// Mitsubishi GX Works2 project: msp_1   PLC: Q03UDV

PROGRAM MAIN
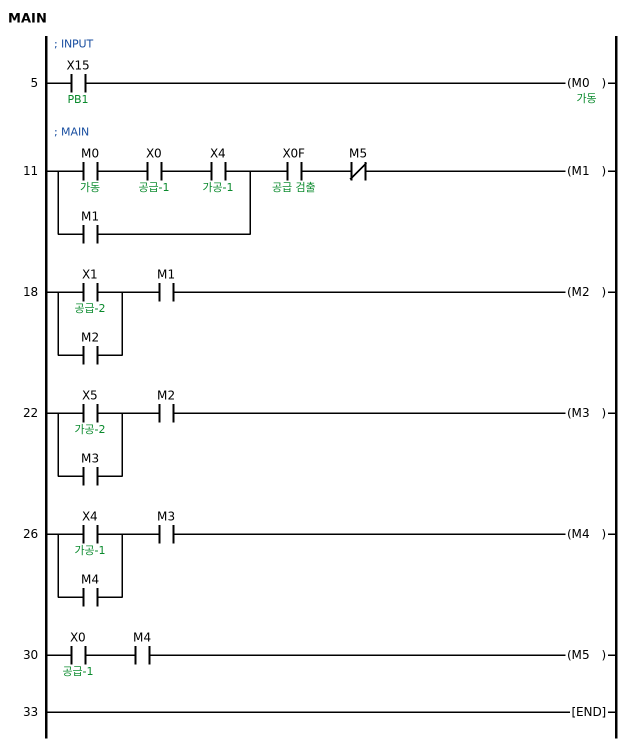
; INPUT
5     LD      X15  ; PB1
      OUT     M0  ; 가동
; MAIN
11    LD      M0  ; 가동
      AND     X0  ; 공급-1
      AND     X4  ; 가공-1
      OR      M1
      AND     X0F  ; 공급 검출
      ANI     M5
      OUT     M1
18    LD      X1  ; 공급-2
      OR      M2
      AND     M1
      OUT     M2
22    LD      X5  ; 가공-2
      OR      M3
      AND     M2
      OUT     M3
26    LD      X4  ; 가공-1
      OR      M4
      AND     M3
      OUT     M4
30    LD      X0  ; 공급-1
      AND     M4
      OUT     M5
33    END
END_PROGRAM

PROGRAM OUTPUT
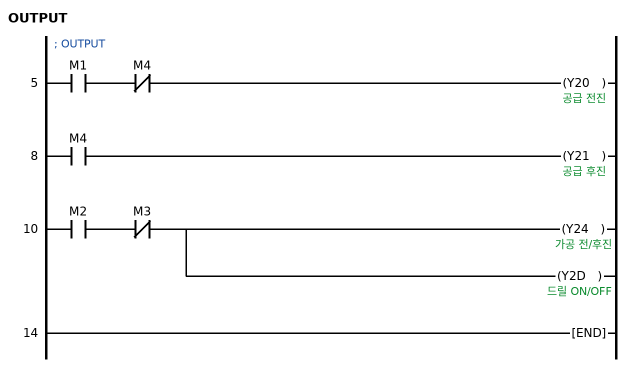
; OUTPUT
5     LD      M1
      ANI     M4
      OUT     Y20  ; 공급 전진
8     LD      M4
      OUT     Y21  ; 공급 후진
10    LD      M2
      ANI     M3
      OUT     Y24  ; 가공 전/후진
      OUT     Y2D  ; 드릴 ON/OFF
14    END
END_PROGRAM

// device comments not shown above
X2  ; 분배-1
X3  ; 분배-2
X6  ; 배출-1
X7  ; 배출-2
X8  ; 스토퍼-1
X9  ; 스토퍼-2
X0A  ; 흡착-1
X0B  ; 흡착-2
X0C  ; 흡착 검출
X0D  ; 창고-1
X0E  ; 창고-2
X10  ; 공급 검출
X11  ; 용량형 센서
X12  ; 유도형 센서
X13  ; 스토퍼 감지
X14  ; 컨벨 인코더
X16  ; PB2
X17  ; PB3
X18  ; PB4
X19  ; PB5
X1A  ; PB6
X1B  ; PB7
X1C  ; PB8
X20  ; A 전진
X21  ; A 후진
X24  ; B 전진/후진
X2D  ; 가공 모터
M14  ; B+
M15  ; B-
M21  ; B+
M22  ; B-
M24  ; A+
M25  ; A-
Y22  ; 분배 전진
Y23  ; 분배 후진
Y25  ; 배출 전진
Y26  ; 배출 후진
Y27  ; 스토퍼 전/후진
Y28  ; 흡착 전진
Y29  ; 흡착 후진
Y2A  ; 흡착 ON/OFF
Y2B  ; 창고 전진
Y2C  ; 창고 후진
Y2E  ; 컨벨 ON/OFF
Y30  ; 램프1
Y31  ; 램프2
Y32  ; 램프3
Y33  ; 램프4
Y34  ; 램프5
Y35  ; 램프6
Y36  ; 램프7
Y37  ; 부저
